(* IEC 61131-3 sources: industrial-data-collection/plc_program, 5 files *)

(* ---- GVL_Config.st ---- *)
// 全局变量列表 - 配置参数
VAR_GLOBAL CONSTANT
    // ========== 传送带配置 ==========
    CONVEYOR_MIN_SPEED: REAL := 0.0;         // 最小速度 (m/s)
    CONVEYOR_MAX_SPEED: REAL := 5.0;         // 最大速度 (m/s)
    CONVEYOR_BASE_POWER: REAL := 0.5;        // 基础功率 (kW)
    CONVEYOR_SPEED_COEFF: REAL := 0.3;       // 速度系数 (kW/(m/s))

    // ========== 工位配置 ==========
    STATION_ACTIVE_POWER: REAL := 5.0;       // 工位运行功率 (kW)
    STATION_STANDBY_POWER: REAL := 0.2;      // 工位待机功率 (kW)
    STATION_PROCESS_TIME: TIME := T#5s;      // 工位加工时间

    // ========== 质量检测配置 ==========
    QUALITY_CHECK_TIME: TIME := T#1s;        // 质量检测时间
    REJECT_ACTIVATE_TIME: TIME := T#2s;      // 剔除机构动作时间

    // ========== 能源计量配置 ==========
    ENERGY_UPDATE_CYCLE: TIME := T#1s;       // 能耗更新周期
    POWER_ALARM_THRESHOLD: REAL := 15.0;     // 功率报警阈值 (kW)

    // ========== 系统配置 ==========
    SYSTEM_SCAN_TIME: TIME := T#100ms;       // 系统扫描时间
END_VAR

(* ---- FB_ConveyorControl.st ---- *)
FUNCTION_BLOCK FB_ConveyorControl
VAR_INPUT
    bStart: BOOL;                    // 启动命令
    rSpeedSetpoint: REAL;            // 速度设定值 (m/s)
    bEmergencyStop: BOOL;            // 紧急停止
END_VAR

VAR_OUTPUT
    bRunning: BOOL;                  // 运行状态
    rActualSpeed: REAL;              // 实际速度 (m/s)
    rPower: REAL;                    // 功率消耗 (kW)
    bFault: BOOL;                    // 故障标志
END_VAR

VAR
    // 内部状态变量
    eState: INT := 0;                // 状态: 0=停止, 1=启动中, 2=运行, 3=停止中
    rCurrentSpeed: REAL := 0.0;      // 当前速度
    rTargetSpeed: REAL := 0.0;       // 目标速度

    // 加减速控制
    rAcceleration: REAL := 0.5;      // 加速度 (m/s²)
    rDeceleration: REAL := 0.8;      // 减速度 (m/s²)
    tScanTime: TIME := T#100ms;      // 扫描时间
    rScanTimeSec: REAL := 0.1;       // 扫描时间(秒)

    // 功率计算参数
    rBasePower: REAL := 0.5;         // 基础功率 (kW)
    rSpeedCoeff: REAL := 0.3;        // 速度系数 (kW/(m/s))

    // 速度限制
    rMinSpeed: REAL := 0.0;          // 最小速度
    rMaxSpeed: REAL := 5.0;          // 最大速度

    // 定时器
    tonStartDelay: TON;              // 启动延时
    tonStopDelay: TON;               // 停止延时

    // 故障检测
    bOverspeed: BOOL := FALSE;       // 超速故障
END_VAR

// ========== 主控制逻辑 ==========

// 紧急停止处理
IF bEmergencyStop THEN
    eState := 0;
    rCurrentSpeed := 0.0;
    rTargetSpeed := 0.0;
    bRunning := FALSE;
    bFault := TRUE;
    RETURN;
END_IF

// 速度设定值限制
rTargetSpeed := LIMIT(rMinSpeed, rSpeedSetpoint, rMaxSpeed);

// 状态机
CASE eState OF
    0: // 停止状态
        rCurrentSpeed := 0.0;
        bRunning := FALSE;
        bFault := FALSE;

        IF bStart AND NOT bEmergencyStop THEN
            eState := 1; // 进入启动状态
            tonStartDelay(IN := FALSE); // 复位定时器
        END_IF

    1: // 启动中
        tonStartDelay(IN := TRUE, PT := T#500ms);

        IF tonStartDelay.Q THEN
            eState := 2; // 进入运行状态
            tonStartDelay(IN := FALSE);
        END_IF

        IF NOT bStart THEN
            eState := 0; // 返回停止状态
        END_IF

    2: // 运行状态
        bRunning := TRUE;

        // 速度控制 - 加速
        IF rCurrentSpeed < rTargetSpeed THEN
            rCurrentSpeed := rCurrentSpeed + (rAcceleration * rScanTimeSec);
            IF rCurrentSpeed > rTargetSpeed THEN
                rCurrentSpeed := rTargetSpeed;
            END_IF
        END_IF

        // 速度控制 - 减速
        IF rCurrentSpeed > rTargetSpeed THEN
            rCurrentSpeed := rCurrentSpeed - (rDeceleration * rScanTimeSec);
            IF rCurrentSpeed < rTargetSpeed THEN
                rCurrentSpeed := rTargetSpeed;
            END_IF
        END_IF

        // 超速检测
        IF rCurrentSpeed > rMaxSpeed THEN
            bOverspeed := TRUE;
            bFault := TRUE;
            eState := 3; // 进入停止状态
        END_IF

        // 停止命令
        IF NOT bStart THEN
            eState := 3; // 进入停止中状态
        END_IF

    3: // 停止中
        bRunning := FALSE;

        // 减速停止
        IF rCurrentSpeed > 0.0 THEN
            rCurrentSpeed := rCurrentSpeed - (rDeceleration * rScanTimeSec);
            IF rCurrentSpeed < 0.0 THEN
                rCurrentSpeed := 0.0;
            END_IF
        ELSE
            eState := 0; // 返回停止状态
            bOverspeed := FALSE;
        END_IF

END_CASE

// ========== 功率计算 ==========
// 功率 = 基础功率 + 速度系数 * 速度
IF bRunning AND rCurrentSpeed > 0.0 THEN
    rPower := rBasePower + (rSpeedCoeff * rCurrentSpeed);
ELSE
    rPower := 0.0;
END_IF

// ========== 输出更新 ==========
rActualSpeed := rCurrentSpeed;

END_FUNCTION_BLOCK

(* ---- FB_EnergyMeter.st ---- *)
FUNCTION_BLOCK FB_EnergyMeter
VAR_INPUT
    bEnable: BOOL;                   // 计量使能
    rPower1: REAL;                   // 设备1功率 (kW)
    rPower2: REAL;                   // 设备2功率 (kW)
    rPower3: REAL;                   // 设备3功率 (kW)
    rPowerThreshold: REAL := 15.0;   // 功率报警阈值 (kW)
    bReset: BOOL;                    // 复位累计能耗
END_VAR

VAR_OUTPUT
    rTotalPower: REAL;               // 总功率 (kW)
    rTotalEnergy: REAL;              // 累计能耗 (kWh)
    rAveragePower: REAL;             // 平均功率 (kW)
    rPeakPower: REAL;                // 峰值功率 (kW)
    bPowerAlarm: BOOL;               // 功率报警
    bDataUpdated: BOOL;              // 数据更新标志
END_VAR

VAR
    // 内部计量变量
    rAccumulatedEnergy: REAL := 0.0; // 累计能耗内部值
    rPowerSum: REAL := 0.0;          // 功率累加和
    iPowerSamples: DINT := 0;        // 功率采样次数
    rPeakPowerInternal: REAL := 0.0; // 峰值功率内部值

    // 定时器
    tonUpdateCycle: TON;             // 更新周期定时器
    tUpdateCycle: TIME := T#1s;      // 更新周期（1秒）

    // 时间计算
    tLastUpdate: TIME;               // 上次更新时间
    tCurrentTime: TIME;              // 当前时间
    tElapsedTime: TIME;              // 经过时间
    rElapsedHours: REAL;             // 经过时间（小时）

    // 扫描时间
    tScanTime: TIME := T#100ms;      // 系统扫描时间
    rScanTimeHours: REAL := 0.0000277778; // 扫描时间（小时）= 100ms / 3600000ms

    // 内部标志
    bFirstScan: BOOL := TRUE;        // 首次扫描标志
    bResetOld: BOOL := FALSE;        // 复位信号旧值
    bResetRising: BOOL := FALSE;     // 复位上升沿

    // 报警相关
    iAlarmCounter: INT := 0;         // 报警计数器
    iAlarmThreshold: INT := 3;       // 连续超阈值次数才报警

    // 数据更新标志
    bUpdateFlag: BOOL := FALSE;      // 内部更新标志
END_VAR

// ========== 主控制逻辑 ==========

// 复位边沿检测
bResetRising := bReset AND NOT bResetOld;
bResetOld := bReset;

// 复位处理
IF bResetRising THEN
    rAccumulatedEnergy := 0.0;
    rPowerSum := 0.0;
    iPowerSamples := 0;
    rPeakPowerInternal := 0.0;
    bPowerAlarm := FALSE;
    iAlarmCounter := 0;
    bFirstScan := TRUE;
END_IF

// 如果未使能，清零输出
IF NOT bEnable THEN
    rTotalPower := 0.0;
    rTotalEnergy := 0.0;
    rAveragePower := 0.0;
    rPeakPower := 0.0;
    bPowerAlarm := FALSE;
    bDataUpdated := FALSE;
    bFirstScan := TRUE;
    RETURN;
END_IF

// ========== 实时功率计算 ==========
// 累加所有设备功率
rTotalPower := rPower1 + rPower2 + rPower3;

// 确保功率为非负值
IF rTotalPower < 0.0 THEN
    rTotalPower := 0.0;
END_IF

// ========== 能耗累计计算 ==========
// 能耗 += 功率 * 时间间隔
// 使用扫描时间作为时间间隔
IF NOT bFirstScan THEN
    // 能耗累计：kWh = kW * hours
    rAccumulatedEnergy := rAccumulatedEnergy + (rTotalPower * rScanTimeHours);
END_IF

// ========== 统计数据计算 ==========
// 功率累加（用于平均值计算）
rPowerSum := rPowerSum + rTotalPower;
iPowerSamples := iPowerSamples + 1;

// 平均功率计算
IF iPowerSamples > 0 THEN
    rAveragePower := rPowerSum / DINT_TO_REAL(iPowerSamples);
ELSE
    rAveragePower := 0.0;
END_IF

// 峰值功率更新
IF rTotalPower > rPeakPowerInternal THEN
    rPeakPowerInternal := rTotalPower;
END_IF

// ========== 异常用电检测 ==========
// 功率超过阈值时设置报警标志
// 使用连续超阈值判定，避免瞬时波动误报
IF rTotalPower > rPowerThreshold THEN
    iAlarmCounter := iAlarmCounter + 1;
    IF iAlarmCounter >= iAlarmThreshold THEN
        bPowerAlarm := TRUE;
    END_IF
ELSE
    iAlarmCounter := 0;
    // 功率恢复正常后，报警需要手动复位或自动清除
    IF rTotalPower < (rPowerThreshold * 0.9) THEN
        bPowerAlarm := FALSE;
    END_IF
END_IF

// ========== 数据更新周期控制 ==========
// 每1秒更新一次数据标志
tonUpdateCycle(IN := TRUE, PT := tUpdateCycle);

IF tonUpdateCycle.Q THEN
    tonUpdateCycle(IN := FALSE); // 复位定时器
    bUpdateFlag := TRUE;
ELSE
    bUpdateFlag := FALSE;
END_IF

// ========== 输出更新 ==========
rTotalEnergy := rAccumulatedEnergy;
rPeakPower := rPeakPowerInternal;
bDataUpdated := bUpdateFlag;

// 清除首次扫描标志
IF bFirstScan THEN
    bFirstScan := FALSE;
END_IF

END_FUNCTION_BLOCK

(* ---- PLC_PRG_MINIMAL.st ---- *)
PROGRAM PLC_PRG_MINIMAL
VAR
    // 最小化测试变量
    bTest: BOOL := FALSE;
    iTest: INT := 0;
    rTest: REAL := 0.0;
END_VAR

// 最简单的逻辑
IF bTest THEN
    iTest := iTest + 1;
    rTest := rTest + 1.0;
END_IF

END_PROGRAM

(* ---- PLC_PRG_SIMPLE_FLOW.st ---- *)
// 简化版产品流动逻辑 - 直接替换PLC_PRG.st中的产品流动部分

// 自动产品流动：简化版本，不使用复杂状态机
IF bAutoMode AND eSystemState = 1 THEN
    // 简单的产品流动：直接模拟产品在两个工位之间流动

    // 工位1：如果没有产品且工位1空闲，生成新产品
    IF NOT bProductSensor1 AND NOT bStation1Processing THEN
        tonProductFlow(IN := TRUE, PT := T#2s);
        IF tonProductFlow.Q THEN
            bProductSensor1 := TRUE;
            iProductGenCounter := iProductGenCounter + 1;
            // 设置质量（90%合格）
            IF iProductGenCounter MOD 10 = 0 THEN
                bQualitySensor := FALSE;
            ELSE
                bQualitySensor := TRUE;
            END_IF
            tonProductFlow(IN := FALSE);
        END_IF
    END_IF

    // 工位1完成后，移动到工位2
    IF bStation1ProcessComplete AND bProductSensor1 AND NOT bProductSensor2 THEN
        tonProductFlow(IN := TRUE, PT := T#2s);
        IF tonProductFlow.Q THEN
            bProductSensor1 := FALSE;
            bProductSensor2 := TRUE;
            tonProductFlow(IN := FALSE);
        END_IF
    END_IF

    // 工位2完成后，触发质量检测
    IF bStation2ProcessComplete AND bProductSensor2 AND NOT bTriggerQualityCheck THEN
        bTriggerQualityCheck := TRUE;
    END_IF

    // 质量检测完成后，产品离开
    IF bQualityCheckComplete AND bProductSensor2 THEN
        tonProductFlow(IN := TRUE, PT := T#2s);
        IF tonProductFlow.Q THEN
            bProductSensor2 := FALSE;
            bTriggerQualityCheck := FALSE;
            tonProductFlow(IN := FALSE);
        END_IF
    END_IF

ELSE
    // 系统停止时复位
    bProductSensor1 := FALSE;
    bProductSensor2 := FALSE;
    bTriggerQualityCheck := FALSE;
    tonProductFlow(IN := FALSE);
END_IF
